TYPE T_PositiveINT : INT(0..32767); END_TYPE

(* stored: Version 1.1.0.1
   DUT T_PositiveINT: Id {b4b075a2-7bff-4795-99b4-fafa6bb84d6e} *)
